SUBAPPLICATION ZaehlerVergleich (* Subapplication Type *)
  (* Standard: 61499-2 *)
  (* Version 1.0, 2023-02-18, Franz *)
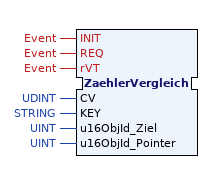
  EVENT_INPUT
    INIT; (* Initialization Request *)
    REQ; (* Normal Execution Request *)
    rVT; (* refresh VT *)
  END_EVENT
  VAR_INPUT
    CV : UDINT; (* Counter Value *)
    KEY : STRING;
    u16ObjId_Ziel : UINT;
    u16ObjId_Pointer : UINT;
  END_VAR
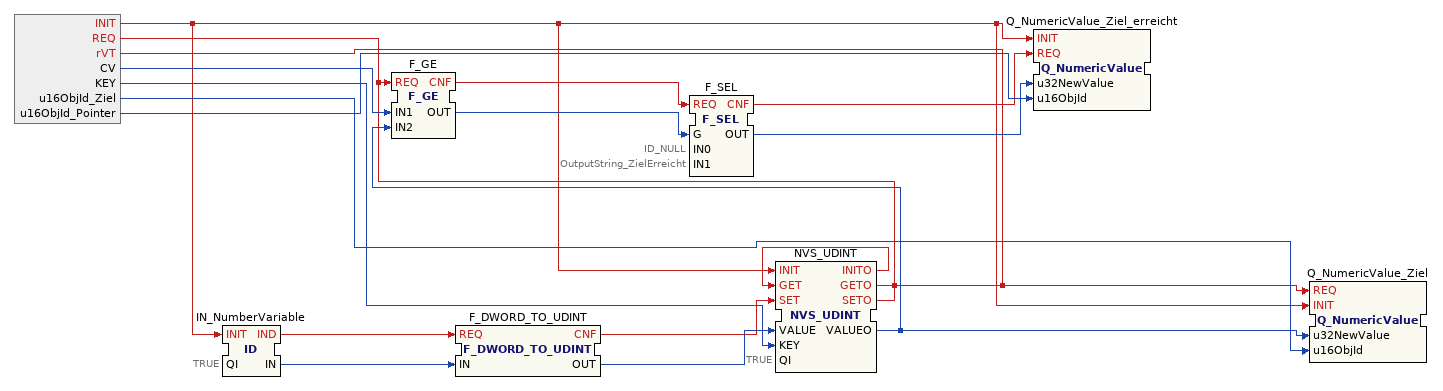
  FBS
    Q_NumericValue_Ziel_erreicht : Q_NumericValue;
    F_GE : F_GE;
    NVS_UDINT : NVS_UDINT(QI := TRUE);
    Q_NumericValue_Ziel : Q_NumericValue;
    F_SEL : F_SEL(IN0 := ID_NULL, IN1 := OutputString_ZielErreicht);
    IN_NumberVariable : ID(QI := TRUE);
    F_DWORD_TO_UDINT : F_DWORD_TO_UDINT;
  END_FBS
  EVENT_CONNECTIONS
    INIT TO Q_NumericValue_Ziel_erreicht.INIT;
    REQ TO F_GE.REQ;
    INIT TO NVS_UDINT.INIT;
    NVS_UDINT.INITO TO NVS_UDINT.GET;
    NVS_UDINT.GETO TO Q_NumericValue_Ziel.REQ;
    INIT TO Q_NumericValue_Ziel.INIT;
    NVS_UDINT.GETO TO F_GE.REQ;
    NVS_UDINT.SETO TO F_GE.REQ;
    rVT TO Q_NumericValue_Ziel.REQ;
    F_GE.CNF TO F_SEL.REQ;
    F_SEL.CNF TO Q_NumericValue_Ziel_erreicht.REQ;
    INIT TO IN_NumberVariable.INIT;
    IN_NumberVariable.IND TO F_DWORD_TO_UDINT.REQ;
    F_DWORD_TO_UDINT.CNF TO NVS_UDINT.SET;
  END_CONNECTIONS
  DATA_CONNECTIONS
    CV TO F_GE.IN1;
    NVS_UDINT.VALUEO TO Q_NumericValue_Ziel.u32NewValue;
    NVS_UDINT.VALUEO TO F_GE.IN2;
    F_GE.OUT TO F_SEL.G;
    F_SEL.OUT TO Q_NumericValue_Ziel_erreicht.u32NewValue;
    IN_NumberVariable.IN TO F_DWORD_TO_UDINT.IN;
    F_DWORD_TO_UDINT.OUT TO NVS_UDINT.VALUE;
    KEY TO NVS_UDINT.KEY;
    u16ObjId_Ziel TO Q_NumericValue_Ziel.u16ObjId;
    u16ObjId_Pointer TO Q_NumericValue_Ziel_erreicht.u16ObjId;
  END_CONNECTIONS
END_SUBAPPLICATION
